// TIA Portal V20 export
// export: Created 2025-12-01T14:57:45.6134644Z, ExportSetting None, DisplayName Totally Integrated Automation Portal, DisplayVersion V20 Update 3, DisplayName TIA Portal Openness, DisplayVersion V20 Update 3, DisplayName TIA Portal Version Control Interface, DisplayVersion V20 Update 3, DisplayName STEP 7 Professional, DisplayVersion V20 Update 3, DisplayName STEP 7 Safety, DisplayVersion V20 Update 2, DisplayName WinCC Basic/Comfort/Advanced, DisplayVersion V20 Update 3, DisplayName WinCC Professional, DisplayVersion V20 Update 3, DisplayName WinCC Unified, DisplayVersion V20 Update 3
FUNCTION_BLOCK "FB420_MesaTL_EtiquetaOrden"   // FB420, LAD
{ S7_Optimized_Access := 'FALSE' }
AUTHOR : ROUTER
NAME : 20180615
VERSION : 3.1
// stored: AutoNumber false, SetENOAutomatically false
   VAR_INPUT
      NumeroMesa : UInt;
      pHsMx : Bool;
      NumSCR : UInt;   // Numero de Scanner asociada a la mesa
      DBFIFO_SCR : UInt;   // DB de Etiquetas Leidas
      LongFIFO_SCR : UInt;   // Numero de Lecturas que se pueden Almacenar
      V_TmpEntrada : Time := T#500MS;
      V_TmpSalida : Time := T#1S;
      MesaDeJDT02 : Bool;
   END_VAR
   VAR_OUTPUT
      PermisoEntrada : Bool;
      PermisoSalida : Bool;
   END_VAR
   VAR
      Mx_ET00 : Bool;
      Mx_ET01 : Bool;
      Mx_ET02 : Bool;
      Mx_ET07 : Bool;
      Mx_ET10 : Bool;
      Mx_ET11 : Bool;
      Mx_ET12 : Bool;
      Mx_ET50 : Bool;
      Mx_ET51 : Bool;
      Mx_ET52 : Bool;
      PresenciaEmiOK : Bool;
      AusenciaEmiOK : Bool;
      BorradoOK : Bool;
      OrdenMx : UInt;
      Motivo : UInt;
      TmpEntrada { S7_SetPoint := 'True'} : TON_TIME;
      TmpSalida { S7_SetPoint := 'True'} : TON_TIME;
      Datos_Scanner { S7_SetPoint := 'True'} : "ROUT_Orden_Fifo_Scanner";
   END_VAR
   VAR_TEMP
      Aux_ET00 : Bool;
      ExisteOrdenSCR : Bool;
      SinOrdenSCR : Bool;
      ExisteOrdenMx : Bool;
      SinOrdenMx : Bool;
      Presencia : Bool;
      Ausencia : Bool;
      Ausencia_especial : Bool;
      MirarOrden : Bool;
      BorradoOrden : Bool;
      Emi_presencia : Bool;
      Emi_ausencia : Bool;
      MesaTMP : UInt;
      MotivoTMP : UInt;
      posicion : Int;
      i : Int;
      longitud : Int;
      codigo_string : String[20];
      mesa_string : String[5];
      moti_string : String[4];
      Mensaje_completo : String;
   END_VAR
BEGIN

REGION Network 1: Incializaciones de la Función
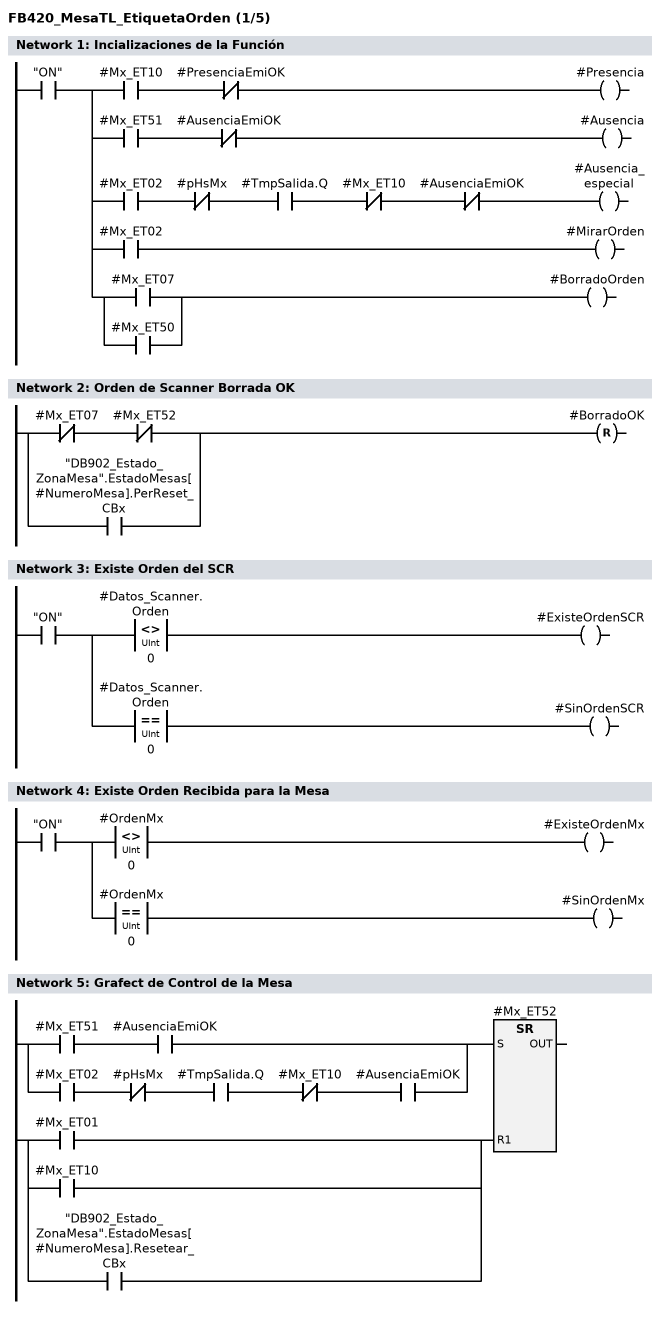
   RUNG wire#powerrail
      Contact( "ON" )
      wire#w1
      Contact( #Mx_ET10 )
      I_Contact( #PresenciaEmiOK )
      Coil( #Presencia )
   END_RUNG
   RUNG wire#w1
      Contact( #Mx_ET51 )
      I_Contact( #AusenciaEmiOK )
      Coil( #Ausencia )
   END_RUNG
   RUNG wire#w1
      Contact( #Mx_ET02 )
      I_Contact( #pHsMx )
      Contact( #TmpSalida.Q )
      I_Contact( #Mx_ET10 )
      I_Contact( #AusenciaEmiOK )
      Coil( #Ausencia_especial )
   END_RUNG
   RUNG wire#w1
      Contact( #Mx_ET02 )
      Coil( #MirarOrden )
   END_RUNG
   RUNG wire#w1
      Contact( #Mx_ET07 )
      wire#w2
      Coil( #BorradoOrden )
   END_RUNG
   RUNG wire#w1
      Contact( #Mx_ET50 )
   END_RUNG wire#w2
   // the same network as SCL:
   #Presencia := "ON" AND #Mx_ET10 AND NOT #PresenciaEmiOK;
   #Ausencia := "ON" AND #Mx_ET51 AND NOT #AusenciaEmiOK;
   #Ausencia_especial := "ON" AND #Mx_ET02 AND NOT #pHsMx AND #TmpSalida.Q AND NOT #Mx_ET10 AND NOT #AusenciaEmiOK;
   #MirarOrden := "ON" AND #Mx_ET02;
   #BorradoOrden := "ON" AND (#Mx_ET07 OR #Mx_ET50);
END_REGION

REGION Network 2: Orden de Scanner Borrada OK
   RUNG wire#powerrail
      I_Contact( #Mx_ET07 )
      I_Contact( #Mx_ET52 )
      wire#w1
      R_Coil( #BorradoOK )
   END_RUNG
   RUNG wire#powerrail
      Contact( "DB902_Estado_ZonaMesa".EstadoMesas[#NumeroMesa].PerReset_CBx )
   END_RUNG wire#w1
   // the same network as SCL:
   IF (NOT #Mx_ET07 AND NOT #Mx_ET52) OR "DB902_Estado_ZonaMesa".EstadoMesas[#NumeroMesa].PerReset_CBx THEN
       #BorradoOK := FALSE;
   END_IF;
END_REGION

REGION Network 3: Existe Orden del SCR
   RUNG wire#powerrail
      Contact( "ON" )
      wire#w1
      { S7_Templates := "SrcType := UInt" } NE_Contact(in1 := #Datos_Scanner.Orden, in2 := 0)
      Coil( #ExisteOrdenSCR )
   END_RUNG
   RUNG wire#w1
      { S7_Templates := "SrcType := UInt" } EQ_Contact(in1 := #Datos_Scanner.Orden, in2 := 0)
      Coil( #SinOrdenSCR )
   END_RUNG
   // the same network as SCL:
   #ExisteOrdenSCR := "ON" AND (#Datos_Scanner.Orden <> 0);
   #SinOrdenSCR := "ON" AND (#Datos_Scanner.Orden = 0);
END_REGION

REGION Network 4: Existe Orden Recibida para la Mesa
   RUNG wire#powerrail
      Contact( "ON" )
      wire#w1
      { S7_Templates := "SrcType := UInt" } NE_Contact(in1 := #OrdenMx, in2 := 0)
      Coil( #ExisteOrdenMx )
   END_RUNG
   RUNG wire#w1
      { S7_Templates := "SrcType := UInt" } EQ_Contact(in1 := #OrdenMx, in2 := 0)
      Coil( #SinOrdenMx )
   END_RUNG
   // the same network as SCL:
   #ExisteOrdenMx := "ON" AND (#OrdenMx <> 0);
   #SinOrdenMx := "ON" AND (#OrdenMx = 0);
END_REGION

REGION Network 5: Grafect de Control de la Mesa
   RUNG wire#powerrail
      Contact( #Mx_ET51 )
      Contact( #AusenciaEmiOK )
      wire#w1
      S_SR(operand := #Mx_ET52, r1 := wire#w2)
   END_RUNG
   RUNG wire#powerrail
      Contact( #Mx_ET02 )
      I_Contact( #pHsMx )
      Contact( #TmpSalida.Q )
      I_Contact( #Mx_ET10 )
      Contact( #AusenciaEmiOK )
   END_RUNG wire#w1
   RUNG wire#powerrail
      Contact( #Mx_ET01 )
   END_RUNG wire#w2
   RUNG wire#powerrail
      Contact( #Mx_ET10 )
   END_RUNG wire#w2
   RUNG wire#powerrail
      Contact( "DB902_Estado_ZonaMesa".EstadoMesas[#NumeroMesa].Resetear_CBx )
   END_RUNG wire#w2
   // the same network as SCL:
   IF (#Mx_ET51 AND #AusenciaEmiOK) OR (#Mx_ET02 AND NOT #pHsMx AND #TmpSalida.Q AND NOT #Mx_ET10 AND #AusenciaEmiOK) THEN
       #Mx_ET52 := TRUE;   // SR flip-flop
   END_IF;
   IF #Mx_ET01 OR #Mx_ET10 OR "DB902_Estado_ZonaMesa".EstadoMesas[#NumeroMesa].Resetear_CBx THEN
       #Mx_ET52 := FALSE;
   END_IF;
END_REGION

REGION Network 6
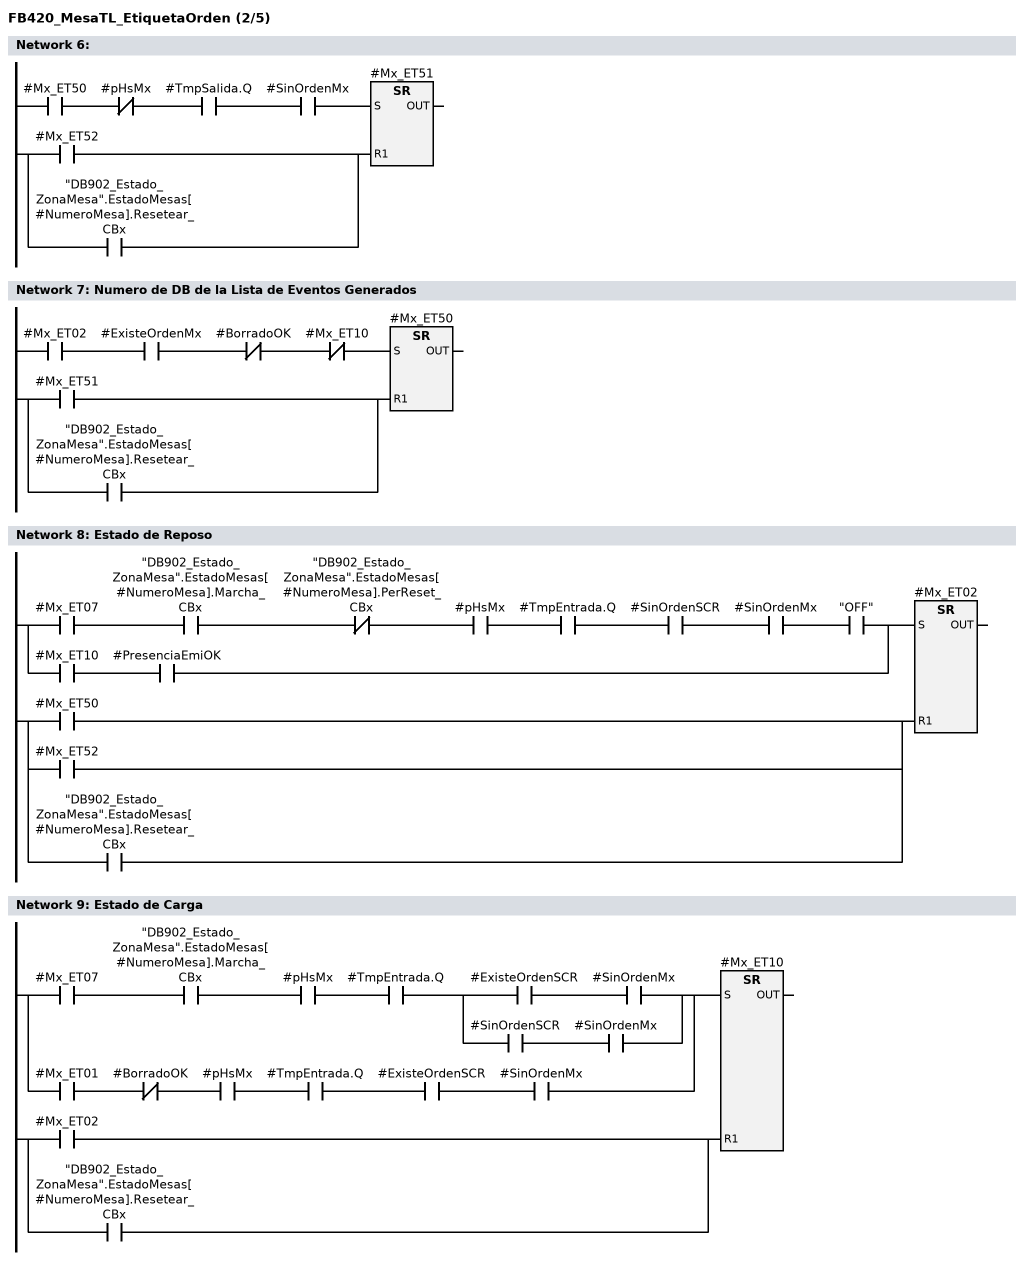
   RUNG wire#powerrail
      Contact( #Mx_ET50 )
      I_Contact( #pHsMx )
      Contact( #TmpSalida.Q )
      Contact( #SinOrdenMx )
      S_SR(operand := #Mx_ET51, r1 := wire#w1)
   END_RUNG
   RUNG wire#powerrail
      Contact( #Mx_ET52 )
   END_RUNG wire#w1
   RUNG wire#powerrail
      Contact( "DB902_Estado_ZonaMesa".EstadoMesas[#NumeroMesa].Resetear_CBx )
   END_RUNG wire#w1
   // the same network as SCL:
   IF #Mx_ET50 AND NOT #pHsMx AND #TmpSalida.Q AND #SinOrdenMx THEN
       #Mx_ET51 := TRUE;   // SR flip-flop
   END_IF;
   IF #Mx_ET52 OR "DB902_Estado_ZonaMesa".EstadoMesas[#NumeroMesa].Resetear_CBx THEN
       #Mx_ET51 := FALSE;
   END_IF;
END_REGION

REGION Network 7: Numero de DB de la Lista de Eventos Generados
   RUNG wire#powerrail
      Contact( #Mx_ET02 )
      Contact( #ExisteOrdenMx )
      I_Contact( #BorradoOK )
      I_Contact( #Mx_ET10 )
      S_SR(operand := #Mx_ET50, r1 := wire#w1)
   END_RUNG
   RUNG wire#powerrail
      Contact( #Mx_ET51 )
   END_RUNG wire#w1
   RUNG wire#powerrail
      Contact( "DB902_Estado_ZonaMesa".EstadoMesas[#NumeroMesa].Resetear_CBx )
   END_RUNG wire#w1
   // the same network as SCL:
   IF #Mx_ET02 AND #ExisteOrdenMx AND NOT #BorradoOK AND NOT #Mx_ET10 THEN
       #Mx_ET50 := TRUE;   // SR flip-flop
   END_IF;
   IF #Mx_ET51 OR "DB902_Estado_ZonaMesa".EstadoMesas[#NumeroMesa].Resetear_CBx THEN
       #Mx_ET50 := FALSE;
   END_IF;
END_REGION

REGION Network 8: Estado de Reposo
   RUNG wire#powerrail
      Contact( #Mx_ET07 )
      Contact( "DB902_Estado_ZonaMesa".EstadoMesas[#NumeroMesa].Marcha_CBx )
      I_Contact( "DB902_Estado_ZonaMesa".EstadoMesas[#NumeroMesa].PerReset_CBx )
      Contact( #pHsMx )
      Contact( #TmpEntrada.Q )
      Contact( #SinOrdenSCR )
      Contact( #SinOrdenMx )
      Contact( "OFF" )
      wire#w1
      S_SR(operand := #Mx_ET02, r1 := wire#w2)
   END_RUNG
   RUNG wire#powerrail
      Contact( #Mx_ET10 )
      Contact( #PresenciaEmiOK )
   END_RUNG wire#w1
   RUNG wire#powerrail
      Contact( #Mx_ET50 )
   END_RUNG wire#w2
   RUNG wire#powerrail
      Contact( #Mx_ET52 )
   END_RUNG wire#w2
   RUNG wire#powerrail
      Contact( "DB902_Estado_ZonaMesa".EstadoMesas[#NumeroMesa].Resetear_CBx )
   END_RUNG wire#w2
   // the same network as SCL:
   IF (#Mx_ET07 AND "DB902_Estado_ZonaMesa".EstadoMesas[#NumeroMesa].Marcha_CBx AND NOT "DB902_Estado_ZonaMesa".EstadoMesas[#NumeroMesa].PerReset_CBx AND #pHsMx AND #TmpEntrada.Q AND #SinOrdenSCR AND #SinOrdenMx AND "OFF") OR (#Mx_ET10 AND #PresenciaEmiOK) THEN
       #Mx_ET02 := TRUE;   // SR flip-flop
   END_IF;
   IF #Mx_ET50 OR #Mx_ET52 OR "DB902_Estado_ZonaMesa".EstadoMesas[#NumeroMesa].Resetear_CBx THEN
       #Mx_ET02 := FALSE;
   END_IF;
END_REGION

REGION Network 9: Estado de Carga
   RUNG wire#powerrail
      Contact( #Mx_ET07 )
      Contact( "DB902_Estado_ZonaMesa".EstadoMesas[#NumeroMesa].Marcha_CBx )
      Contact( #pHsMx )
      Contact( #TmpEntrada.Q )
      wire#w1
      Contact( #ExisteOrdenSCR )
      Contact( #SinOrdenMx )
      wire#w2
      S_SR(operand := #Mx_ET10, r1 := wire#w3)
   END_RUNG
   RUNG wire#w1
      Contact( #SinOrdenSCR )
      Contact( #SinOrdenMx )
   END_RUNG wire#w2
   RUNG wire#powerrail
      Contact( #Mx_ET01 )
      I_Contact( #BorradoOK )
      Contact( #pHsMx )
      Contact( #TmpEntrada.Q )
      Contact( #ExisteOrdenSCR )
      Contact( #SinOrdenMx )
   END_RUNG wire#w2
   RUNG wire#powerrail
      Contact( #Mx_ET02 )
   END_RUNG wire#w3
   RUNG wire#powerrail
      Contact( "DB902_Estado_ZonaMesa".EstadoMesas[#NumeroMesa].Resetear_CBx )
   END_RUNG wire#w3
   // the same network as SCL:
   IF (#Mx_ET07 AND "DB902_Estado_ZonaMesa".EstadoMesas[#NumeroMesa].Marcha_CBx AND #pHsMx AND #TmpEntrada.Q AND ((#ExisteOrdenSCR AND #SinOrdenMx) OR (#SinOrdenSCR AND #SinOrdenMx))) OR (#Mx_ET01 AND NOT #BorradoOK AND #pHsMx AND #TmpEntrada.Q AND #ExisteOrdenSCR AND #SinOrdenMx) THEN
       #Mx_ET10 := TRUE;   // SR flip-flop
   END_IF;
   IF #Mx_ET02 OR "DB902_Estado_ZonaMesa".EstadoMesas[#NumeroMesa].Resetear_CBx THEN
       #Mx_ET10 := FALSE;
   END_IF;
END_REGION

REGION Network 10: Estado de Vacia
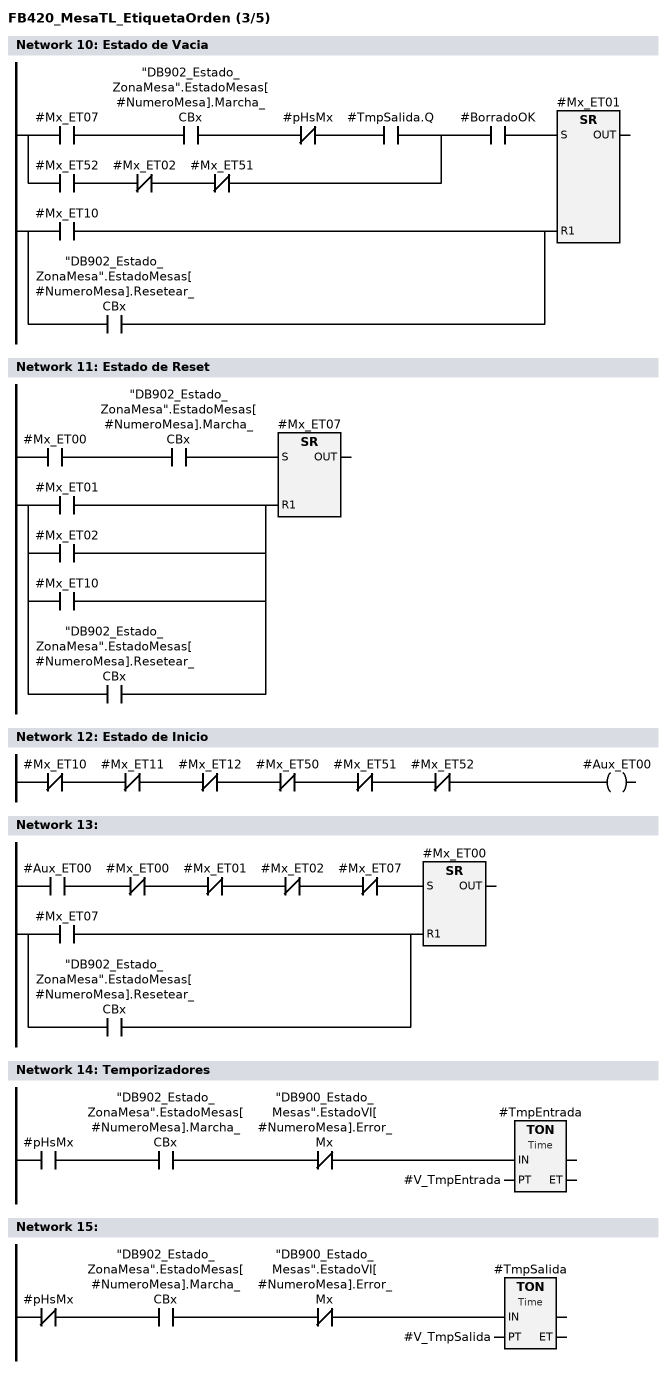
   RUNG wire#powerrail
      Contact( #Mx_ET07 )
      Contact( "DB902_Estado_ZonaMesa".EstadoMesas[#NumeroMesa].Marcha_CBx )
      I_Contact( #pHsMx )
      Contact( #TmpSalida.Q )
      wire#w1
      Contact( #BorradoOK )
      S_SR(operand := #Mx_ET01, r1 := wire#w2)
   END_RUNG
   RUNG wire#powerrail
      Contact( #Mx_ET52 )
      I_Contact( #Mx_ET02 )
      I_Contact( #Mx_ET51 )
   END_RUNG wire#w1
   RUNG wire#powerrail
      Contact( #Mx_ET10 )
   END_RUNG wire#w2
   RUNG wire#powerrail
      Contact( "DB902_Estado_ZonaMesa".EstadoMesas[#NumeroMesa].Resetear_CBx )
   END_RUNG wire#w2
   // the same network as SCL:
   IF ((#Mx_ET07 AND "DB902_Estado_ZonaMesa".EstadoMesas[#NumeroMesa].Marcha_CBx AND NOT #pHsMx AND #TmpSalida.Q) OR (#Mx_ET52 AND NOT #Mx_ET02 AND NOT #Mx_ET51)) AND #BorradoOK THEN
       #Mx_ET01 := TRUE;   // SR flip-flop
   END_IF;
   IF #Mx_ET10 OR "DB902_Estado_ZonaMesa".EstadoMesas[#NumeroMesa].Resetear_CBx THEN
       #Mx_ET01 := FALSE;
   END_IF;
END_REGION

REGION Network 11: Estado de Reset
   RUNG wire#powerrail
      Contact( #Mx_ET00 )
      Contact( "DB902_Estado_ZonaMesa".EstadoMesas[#NumeroMesa].Marcha_CBx )
      S_SR(operand := #Mx_ET07, r1 := wire#w1)
   END_RUNG
   RUNG wire#powerrail
      Contact( #Mx_ET01 )
   END_RUNG wire#w1
   RUNG wire#powerrail
      Contact( #Mx_ET02 )
   END_RUNG wire#w1
   RUNG wire#powerrail
      Contact( #Mx_ET10 )
   END_RUNG wire#w1
   RUNG wire#powerrail
      Contact( "DB902_Estado_ZonaMesa".EstadoMesas[#NumeroMesa].Resetear_CBx )
   END_RUNG wire#w1
   // the same network as SCL:
   IF #Mx_ET00 AND "DB902_Estado_ZonaMesa".EstadoMesas[#NumeroMesa].Marcha_CBx THEN
       #Mx_ET07 := TRUE;   // SR flip-flop
   END_IF;
   IF #Mx_ET01 OR #Mx_ET02 OR #Mx_ET10 OR "DB902_Estado_ZonaMesa".EstadoMesas[#NumeroMesa].Resetear_CBx THEN
       #Mx_ET07 := FALSE;
   END_IF;
END_REGION

REGION Network 12: Estado de Inicio
   RUNG wire#powerrail
      I_Contact( #Mx_ET10 )
      I_Contact( #Mx_ET11 )
      I_Contact( #Mx_ET12 )
      I_Contact( #Mx_ET50 )
      I_Contact( #Mx_ET51 )
      I_Contact( #Mx_ET52 )
      Coil( #Aux_ET00 )
   END_RUNG
   // the same network as SCL:
   #Aux_ET00 := NOT #Mx_ET10 AND NOT #Mx_ET11 AND NOT #Mx_ET12 AND NOT #Mx_ET50 AND NOT #Mx_ET51 AND NOT #Mx_ET52;
END_REGION

REGION Network 13
   RUNG wire#powerrail
      Contact( #Aux_ET00 )
      I_Contact( #Mx_ET00 )
      I_Contact( #Mx_ET01 )
      I_Contact( #Mx_ET02 )
      I_Contact( #Mx_ET07 )
      S_SR(operand := #Mx_ET00, r1 := wire#w1)
   END_RUNG
   RUNG wire#powerrail
      Contact( #Mx_ET07 )
   END_RUNG wire#w1
   RUNG wire#powerrail
      Contact( "DB902_Estado_ZonaMesa".EstadoMesas[#NumeroMesa].Resetear_CBx )
   END_RUNG wire#w1
   // the same network as SCL:
   IF #Aux_ET00 AND NOT #Mx_ET00 AND NOT #Mx_ET01 AND NOT #Mx_ET02 AND NOT #Mx_ET07 THEN
       #Mx_ET00 := TRUE;   // SR flip-flop
   END_IF;
   IF #Mx_ET07 OR "DB902_Estado_ZonaMesa".EstadoMesas[#NumeroMesa].Resetear_CBx THEN
       #Mx_ET00 := FALSE;
   END_IF;
END_REGION

REGION Network 14: Temporizadores
   RUNG wire#powerrail
      Contact( #pHsMx )
      Contact( "DB902_Estado_ZonaMesa".EstadoMesas[#NumeroMesa].Marcha_CBx )
      I_Contact( "DB900_Estado_Mesas".EstadoVI[#NumeroMesa].Error_Mx )
      { S7_Templates := "time_type := Time" } #TmpEntrada.TON(pt := #V_TmpEntrada, et =>)
   END_RUNG
   // the same network as SCL:
   #TmpEntrada(IN := #pHsMx AND "DB902_Estado_ZonaMesa".EstadoMesas[#NumeroMesa].Marcha_CBx AND NOT "DB900_Estado_Mesas".EstadoVI[#NumeroMesa].Error_Mx,   // TON
               PT := #V_TmpEntrada);
END_REGION

REGION Network 15
   RUNG wire#powerrail
      I_Contact( #pHsMx )
      Contact( "DB902_Estado_ZonaMesa".EstadoMesas[#NumeroMesa].Marcha_CBx )
      I_Contact( "DB900_Estado_Mesas".EstadoVI[#NumeroMesa].Error_Mx )
      { S7_Templates := "time_type := Time" } #TmpSalida.TON(pt := #V_TmpSalida, et =>)
   END_RUNG
   // the same network as SCL:
   #TmpSalida(IN := NOT #pHsMx AND "DB902_Estado_ZonaMesa".EstadoMesas[#NumeroMesa].Marcha_CBx AND NOT "DB900_Estado_Mesas".EstadoVI[#NumeroMesa].Error_Mx,   // TON
              PT := #V_TmpSalida);
END_REGION

REGION Network 16: Eliminar la Lectura de Scanner
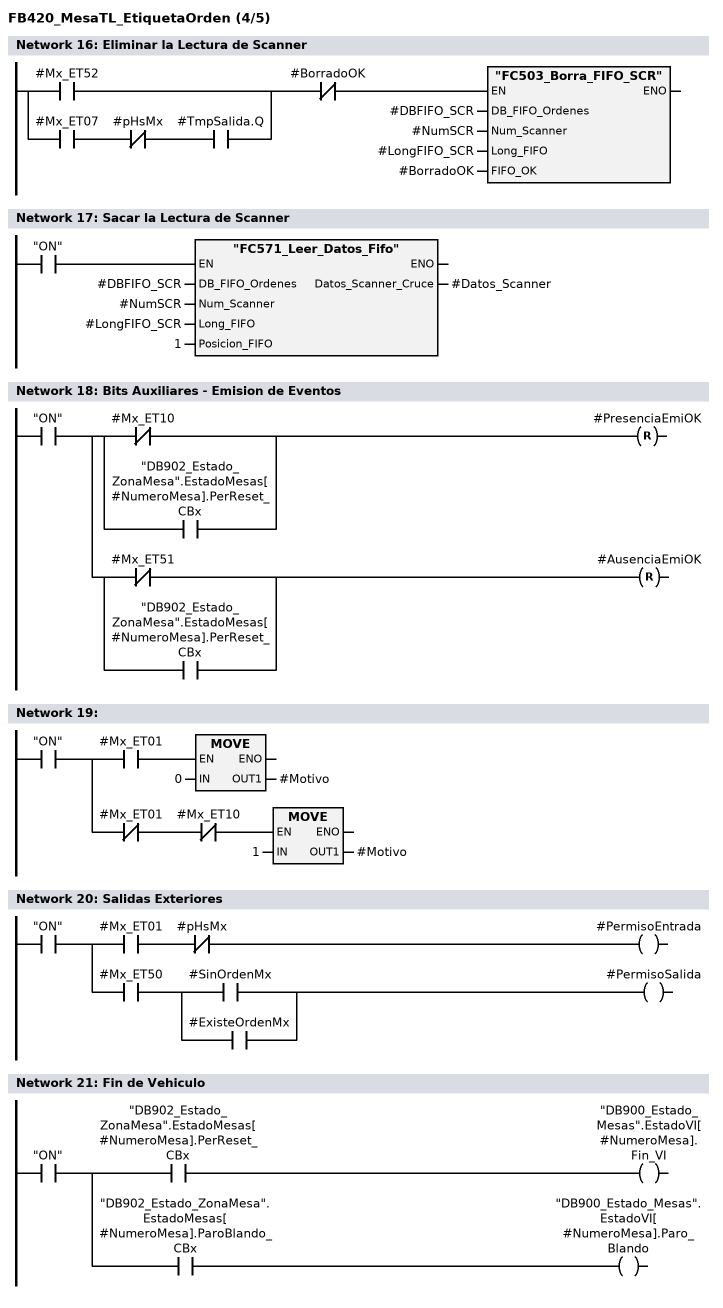
   RUNG wire#powerrail
      Contact( #Mx_ET52 )
      wire#w1
      I_Contact( #BorradoOK )
      "FC503_Borra_FIFO_SCR"(DB_FIFO_Ordenes := #DBFIFO_SCR, Num_Scanner := #NumSCR, Long_FIFO := #LongFIFO_SCR, FIFO_OK := #BorradoOK)
   END_RUNG
   RUNG wire#powerrail
      Contact( #Mx_ET07 )
      I_Contact( #pHsMx )
      Contact( #TmpSalida.Q )
   END_RUNG wire#w1
   // the same network as SCL:
   IF (#Mx_ET52 OR (#Mx_ET07 AND NOT #pHsMx AND #TmpSalida.Q)) AND NOT #BorradoOK THEN
       "FC503_Borra_FIFO_SCR"(DB_FIFO_Ordenes := #DBFIFO_SCR,
                              Num_Scanner := #NumSCR,
                              Long_FIFO := #LongFIFO_SCR,
                              FIFO_OK := #BorradoOK);
   END_IF;
END_REGION

REGION Network 17: Sacar la Lectura de Scanner
   RUNG wire#powerrail
      Contact( "ON" )
      "FC571_Leer_Datos_Fifo"(DB_FIFO_Ordenes := #DBFIFO_SCR, Num_Scanner := #NumSCR, Long_FIFO := #LongFIFO_SCR, Posicion_FIFO := 1, Datos_Scanner_Cruce => #Datos_Scanner)
   END_RUNG
   // the same network as SCL:
   IF "ON" THEN
       "FC571_Leer_Datos_Fifo"(DB_FIFO_Ordenes := #DBFIFO_SCR,
                               Num_Scanner := #NumSCR,
                               Long_FIFO := #LongFIFO_SCR,
                               Posicion_FIFO := 1,
                               Datos_Scanner_Cruce => #Datos_Scanner);
   END_IF;
END_REGION

REGION Network 18: Bits Auxiliares - Emision de Eventos
   RUNG wire#powerrail
      Contact( "ON" )
      wire#w1
      I_Contact( #Mx_ET10 )
      wire#w2
      R_Coil( #PresenciaEmiOK )
   END_RUNG
   RUNG wire#w1
      Contact( "DB902_Estado_ZonaMesa".EstadoMesas[#NumeroMesa].PerReset_CBx )
   END_RUNG wire#w2
   RUNG wire#w1
      I_Contact( #Mx_ET51 )
      wire#w3
      R_Coil( #AusenciaEmiOK )
   END_RUNG
   RUNG wire#w1
      Contact( "DB902_Estado_ZonaMesa".EstadoMesas[#NumeroMesa].PerReset_CBx )
   END_RUNG wire#w3
   // the same network as SCL:
   IF "ON" AND (NOT #Mx_ET10 OR "DB902_Estado_ZonaMesa".EstadoMesas[#NumeroMesa].PerReset_CBx) THEN
       #PresenciaEmiOK := FALSE;
   END_IF;
   IF "ON" AND (NOT #Mx_ET51 OR "DB902_Estado_ZonaMesa".EstadoMesas[#NumeroMesa].PerReset_CBx) THEN
       #AusenciaEmiOK := FALSE;
   END_IF;
END_REGION

REGION Network 19
   RUNG wire#powerrail
      Contact( "ON" )
      wire#w1
      Contact( #Mx_ET01 )
      { S7_GenerateENO := "TRUE" } Move(in := 0, out1 => #Motivo)
   END_RUNG
   RUNG wire#w1
      I_Contact( #Mx_ET01 )
      I_Contact( #Mx_ET10 )
      { S7_GenerateENO := "TRUE" } Move(in := 1, out1 => #Motivo)
   END_RUNG
   // the same network as SCL:
   IF "ON" AND #Mx_ET01 THEN #Motivo := 0; END_IF;
   IF "ON" AND NOT #Mx_ET01 AND NOT #Mx_ET10 THEN #Motivo := 1; END_IF;
END_REGION

REGION Network 20: Salidas Exteriores
   RUNG wire#powerrail
      Contact( "ON" )
      wire#w1
      Contact( #Mx_ET01 )
      I_Contact( #pHsMx )
      Coil( #PermisoEntrada )
   END_RUNG
   RUNG wire#w1
      Contact( #Mx_ET50 )
      wire#w2
      Contact( #SinOrdenMx )
      wire#w3
      Coil( #PermisoSalida )
   END_RUNG
   RUNG wire#w2
      Contact( #ExisteOrdenMx )
   END_RUNG wire#w3
   // the same network as SCL:
   #PermisoEntrada := "ON" AND #Mx_ET01 AND NOT #pHsMx;
   #PermisoSalida := "ON" AND #Mx_ET50 AND (#SinOrdenMx OR #ExisteOrdenMx);
END_REGION

REGION Network 21: Fin de Vehiculo
   RUNG wire#powerrail
      Contact( "ON" )
      wire#w1
      Contact( "DB902_Estado_ZonaMesa".EstadoMesas[#NumeroMesa].PerReset_CBx )
      Coil( "DB900_Estado_Mesas".EstadoVI[#NumeroMesa].Fin_VI )
   END_RUNG
   RUNG wire#w1
      Contact( "DB902_Estado_ZonaMesa".EstadoMesas[#NumeroMesa].ParoBlando_CBx )
      Coil( "DB900_Estado_Mesas".EstadoVI[#NumeroMesa].Paro_Blando )
   END_RUNG
   // the same network as SCL:
   "DB900_Estado_Mesas".EstadoVI[#NumeroMesa].Fin_VI := "ON" AND "DB902_Estado_ZonaMesa".EstadoMesas[#NumeroMesa].PerReset_CBx;
   "DB900_Estado_Mesas".EstadoVI[#NumeroMesa].Paro_Blando := "ON" AND "DB902_Estado_ZonaMesa".EstadoMesas[#NumeroMesa].ParoBlando_CBx;
END_REGION

REGION Network 22
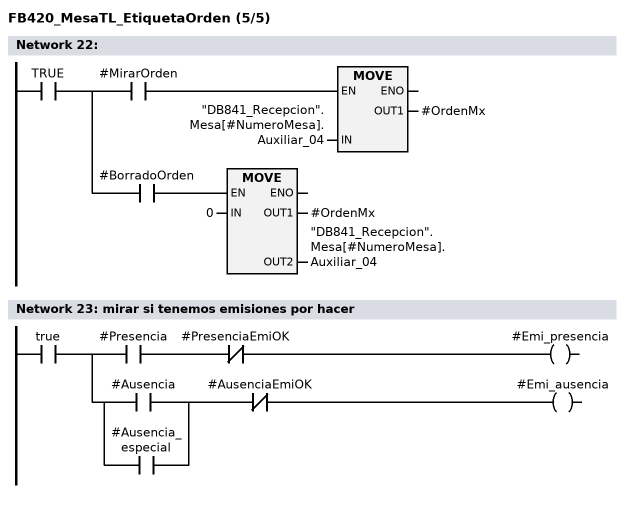
   RUNG wire#powerrail
      Contact( TRUE )
      wire#w1
      Contact( #MirarOrden )
      Move(in := "DB841_Recepcion".Mesa[#NumeroMesa].Auxiliar_04, out1 => #OrdenMx)
   END_RUNG
   RUNG wire#w1
      Contact( #BorradoOrden )
      Move(in := 0, out1 => #OrdenMx, out2 => "DB841_Recepcion".Mesa[#NumeroMesa].Auxiliar_04)
   END_RUNG
   // the same network as SCL:
   IF TRUE AND #MirarOrden THEN #OrdenMx := "DB841_Recepcion".Mesa[#NumeroMesa].Auxiliar_04; END_IF;
   IF TRUE AND #BorradoOrden THEN
       #OrdenMx := 0;
       "DB841_Recepcion".Mesa[#NumeroMesa].Auxiliar_04 := 0;
   END_IF;
END_REGION

REGION Network 23: mirar si tenemos emisiones por hacer
   RUNG wire#powerrail
      Contact( true )
      wire#w1
      Contact( #Presencia )
      I_Contact( #PresenciaEmiOK )
      Coil( #Emi_presencia )
   END_RUNG
   RUNG wire#w1
      Contact( #Ausencia )
      wire#w2
      I_Contact( #AusenciaEmiOK )
      Coil( #Emi_ausencia )
   END_RUNG
   RUNG wire#w1
      Contact( #Ausencia_especial )
   END_RUNG wire#w2
   // the same network as SCL:
   #Emi_presencia := true AND #Presencia AND NOT #PresenciaEmiOK;
   #Emi_ausencia := true AND (#Ausencia OR #Ausencia_especial) AND NOT #AusenciaEmiOK;
END_REGION

REGION Network 24 (SCL)
   IF (#Emi_presencia = true) OR (#Emi_ausencia = true) THEN
       #MesaTMP := #NumeroMesa + "CTE_OffsetMesa";
       #MotivoTMP := #Motivo;
   ELSE
       RETURN;
   END_IF;
END_REGION

REGION Network 25 (SCL)
   //miramos si tenemos que emitir el evento al JDT1 o al JDT2 para buscar hueco
   IF #MesaDeJDT02 = true THEN
   REGION buscar en JDT2

       #posicion := -1;
       FOR #i := 0 TO 100 BY 1 DO
           #longitud := LEN("DB197_eventos_generados_routing_JDT2".evento[#i]);
           IF #longitud = 0 THEN
               #posicion := #i;
               EXIT;
           END_IF;
       END_FOR;

       // si no hay sitio para escribir salimos del bloque
       IF #posicion = -1 THEN
           RETURN;
       END_IF;
   END_REGION
   ;
   ELSE
       REGION buscar en JDT1

           #posicion := -1;
           FOR #i := 0 TO 100 BY 1 DO
               #longitud := LEN("DB198_eventos_generados_routing_JDT1".evento[#i]);
               IF #longitud = 0 THEN
                   #posicion := #i;
                   EXIT;
               END_IF;
           END_FOR;

           // si no hay sitio para escribir salimos del bloque
           IF #posicion = -1 THEN
               RETURN;
           END_IF;
       END_REGION
   END_IF;


   // si continuamos es porque podemos formatear el mensaje
   // 




   #mesa_string := DELETE(IN := (UINT_TO_STRING(IN := #MesaTMP )), L := 1, P := 1);
   #codigo_string := DELETE(IN := (ULINT_TO_STRING(IN := #Datos_Scanner.Identificador)), L := 1, P := 1);

   // CODIFICACION DEL MOTIVO
   #moti_string := '----'; // INICIALIAMOS A ESTE VALOR POR SI ACASO

   IF ((#Emi_presencia=TRUE)AND(#MotivoTMP= 0)) THEN
       #moti_string := 'NORM';
   ELSIF((#Emi_presencia=TRUE)AND(#MotivoTMP= 1)) THEN
       #moti_string := 'RESE';
   ELSIF((#Emi_ausencia=TRUE)AND(#Ausencia_especial=FALSE)) THEN
       #moti_string := 'NORM';
   ELSIF((#Emi_ausencia=TRUE)AND(#Ausencia_especial=TRUE)) THEN
       #moti_string := 'FAIL';
   END_IF;



   // aqui formateamos el mensaje que toca presencia, ausencia o ausencia especial

   IF #Emi_presencia = true THEN
       #Mensaje_completo:= CONCAT(IN1 := '{PRES[MESA]', IN2 := #mesa_string, IN3 := '[SSCC]', IN4 := #codigo_string, IN5 := '[MOTI]', IN6 := #moti_string,IN7:="DB921_DATOS_FECHA_HORA".TIME_STAMP,IN8:='}');
       #PresenciaEmiOK := TRUE;
   ELSIF #Emi_ausencia = TRUE THEN
       #Mensaje_completo := CONCAT(IN1 := '{AUSE[MESA]', IN2 := #mesa_string, IN3 := '[SSCC]', IN4 := #codigo_string, IN5 := '[MOTI]', IN6 := #moti_string,IN7:="DB921_DATOS_FECHA_HORA".TIME_STAMP,IN8:='}');
       #AusenciaEmiOK := TRUE;
   END_IF;

   // ESCRIBIMOS EN EL DB DE EMISIÓN DEL jdt QUE CORRESPONDE
   // 
   IF #MesaDeJDT02 = true THEN

       "DB197_eventos_generados_routing_JDT2".evento[#posicion] := #Mensaje_completo;
   ELSE
       "DB198_eventos_generados_routing_JDT1".evento[#posicion] := #Mensaje_completo;

   END_IF;
END_REGION
END_FUNCTION_BLOCK
